// SIMATIC S7-200 project (STEP 7-Micro/WIN), CPU 226 CN REL 02.01

ORGANIZATION_BLOCK 主程序:OB1
TITLE=程序注释
BEGIN
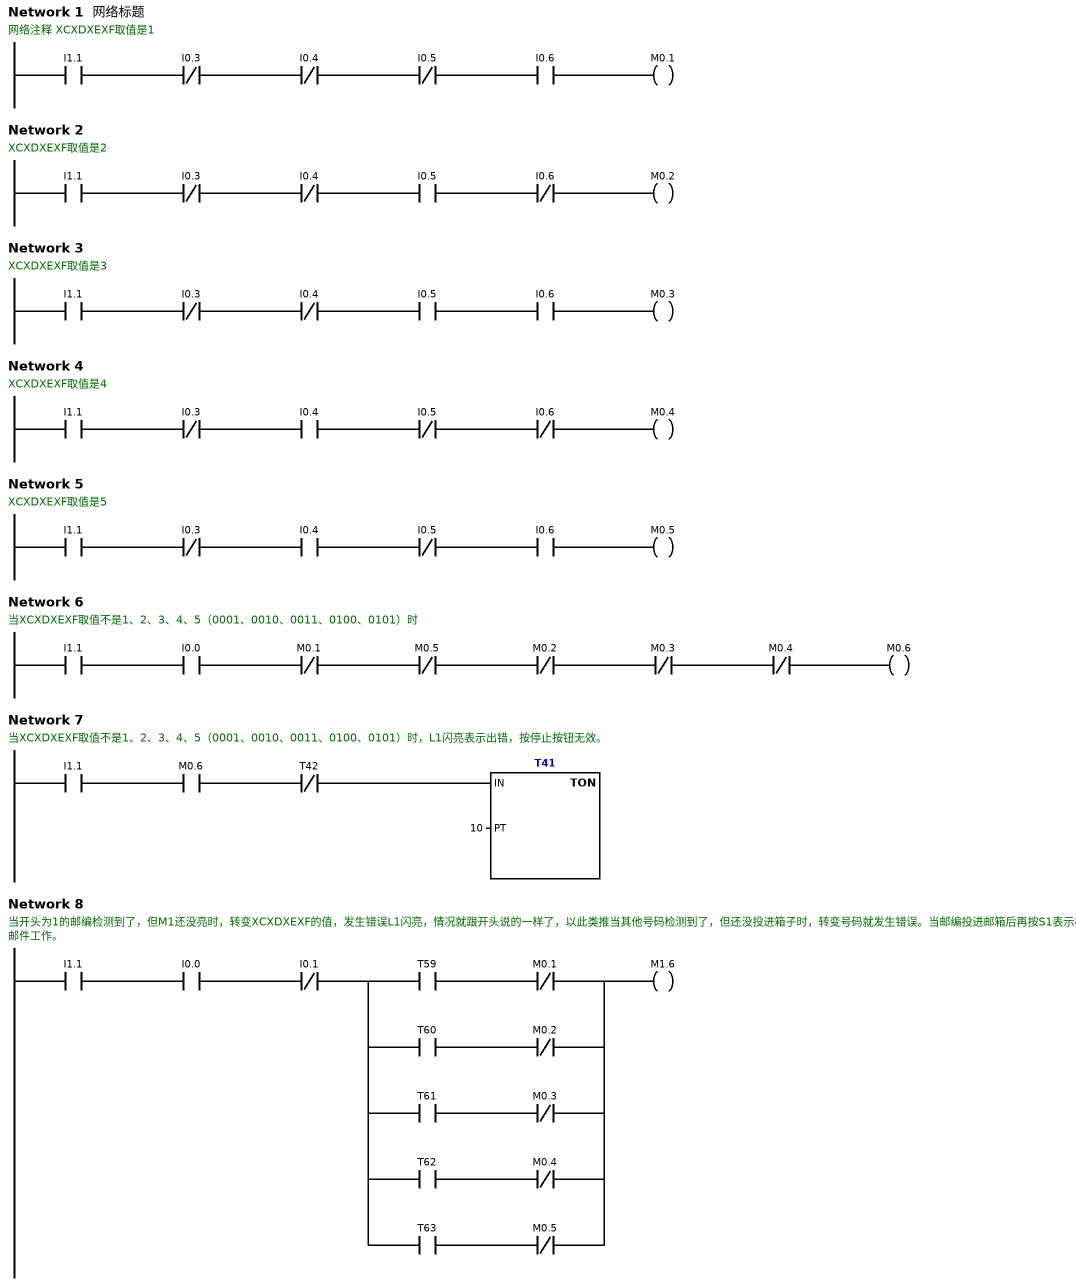
Network 1 // 网络标题
// 网络注释 XCXDXEXF取值是1
LD     I1.1
AN     I0.3
AN     I0.4
AN     I0.5
A      I0.6
=      M0.1
Network 2
// XCXDXEXF取值是2
LD     I1.1
AN     I0.3
AN     I0.4
A      I0.5
AN     I0.6
=      M0.2
Network 3
// XCXDXEXF取值是3
LD     I1.1
AN     I0.3
AN     I0.4
A      I0.5
A      I0.6
=      M0.3
Network 4
// XCXDXEXF取值是4
LD     I1.1
AN     I0.3
A      I0.4
AN     I0.5
AN     I0.6
=      M0.4
Network 5
// XCXDXEXF取值是5
LD     I1.1
AN     I0.3
A      I0.4
AN     I0.5
A      I0.6
=      M0.5
Network 6
// 当XCXDXEXF取值不是1、2、3、4、5（0001、0010、0011、0100、0101）时
LD     I1.1
A      I0.0
AN     M0.1
AN     M0.5
AN     M0.2
AN     M0.3
AN     M0.4
=      M0.6
Network 7
// 当XCXDXEXF取值不是1、2、3、4、5（0001、0010、0011、0100、0101）时，L1闪亮表示出错，按停止按钮无效。
LD     I1.1
A      M0.6
AN     T42
TON    T41, 10
Network 8
// 当开头为1的邮编检测到了，但M1还没亮时，转变XCXDXEXF的值，发生错误L1闪亮，情况就跟开头说的一样了，以此类推当其他号码检测到了，但还没投进箱子时，转变号码就发生错误。当邮编投进邮箱后再按S1表示检测到邮件工作。
// (network saved uncompiled; LAD cells follow)
// row 0: c0 -| |- I1.1  c1 -| |- I0.0  c2 -|/|- I0.1 v  c3 -| |- T59  c4 -|/|- M0.1 v  c5 -( ) M1.6
// row 1: c2 ^v  c3 -| |- T60  c4 -|/|- M0.2 ^v
// row 2: c2 ^v  c3 -| |- T61  c4 -|/|- M0.3 ^v
// row 3: c2 ^v  c3 -| |- T62  c4 -|/|- M0.4 ^v
// row 4: c2 ^  c3 -| |- T63  c4 -|/|- M0.5 ^
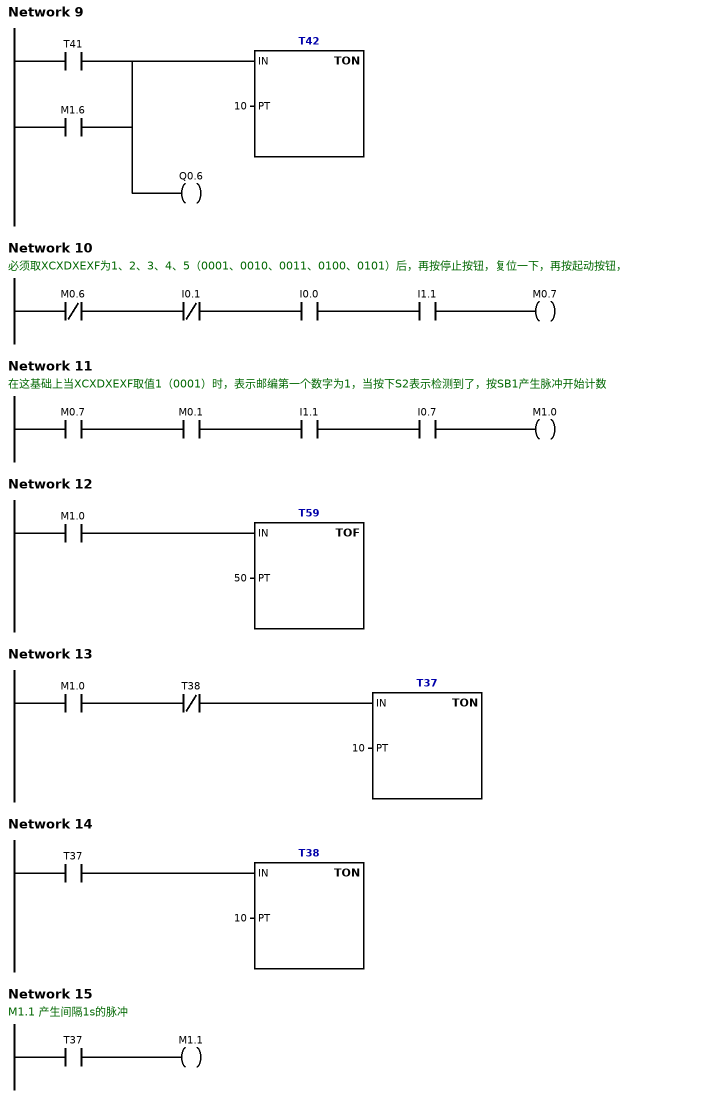
Network 9
LD     T41
O      M1.6
TON    T42, 10
=      Q0.6
Network 10
// 必须取XCXDXEXF为1、2、3、4、5（0001、0010、0011、0100、0101）后，再按停止按钮，复位一下，再按起动按钮，
LDN    M0.6
AN     I0.1
A      I0.0
A      I1.1
=      M0.7
Network 11
// 在这基础上当XCXDXEXF取值1（0001）时，表示邮编第一个数字为1，当按下S2表示检测到了，按SB1产生脉冲开始计数
LD     M0.7
A      M0.1
A      I1.1
A      I0.7
=      M1.0
Network 12
// (network saved uncompiled; LAD cells follow)
// row 0: c0 -| |- M1.0  c1 --  c2 [TOF T59 IN:=power@row0, PT:=50]
// row 1: c2 [box]
Network 13
LD     M1.0
AN     T38
TON    T37, 10
Network 14
LD     T37
TON    T38, 10
Network 15
// M1.1 产生间隔1s的脉冲
LD     T37
=      M1.1
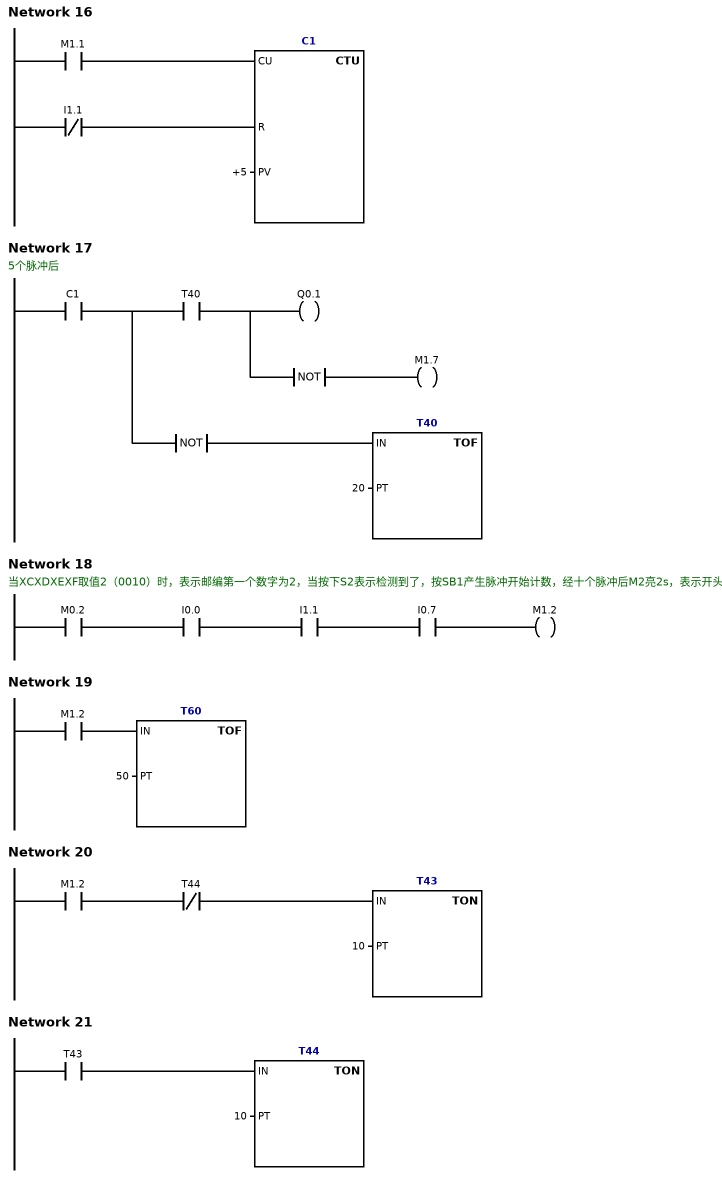
Network 16
LD     M1.1
LDN    I1.1
CTU    C1, +5
Network 17
// 5个脉冲后
LD     C1
LPS
A      T40
=      Q0.1
NOT
=      M1.7
LPP
NOT
TOF    T40, 20
Network 18
// 当XCXDXEXF取值2（0010）时，表示邮编第一个数字为2，当按下S2表示检测到了，按SB1产生脉冲开始计数，经十个脉冲后M2亮2s，表示开头为2的邮编进上海的邮箱，同时M5、L2、S1灭2s。
LD     M0.2
A      I0.0
A      I1.1
A      I0.7
=      M1.2
Network 19
// (network saved uncompiled; LAD cells follow)
// row 0: c0 -| |- M1.2  c1 [TOF T60 IN:=power@row0, PT:=50]
// row 1: c1 [box]
Network 20
LD     M1.2
AN     T44
TON    T43, 10
Network 21
LD     T43
TON    T44, 10
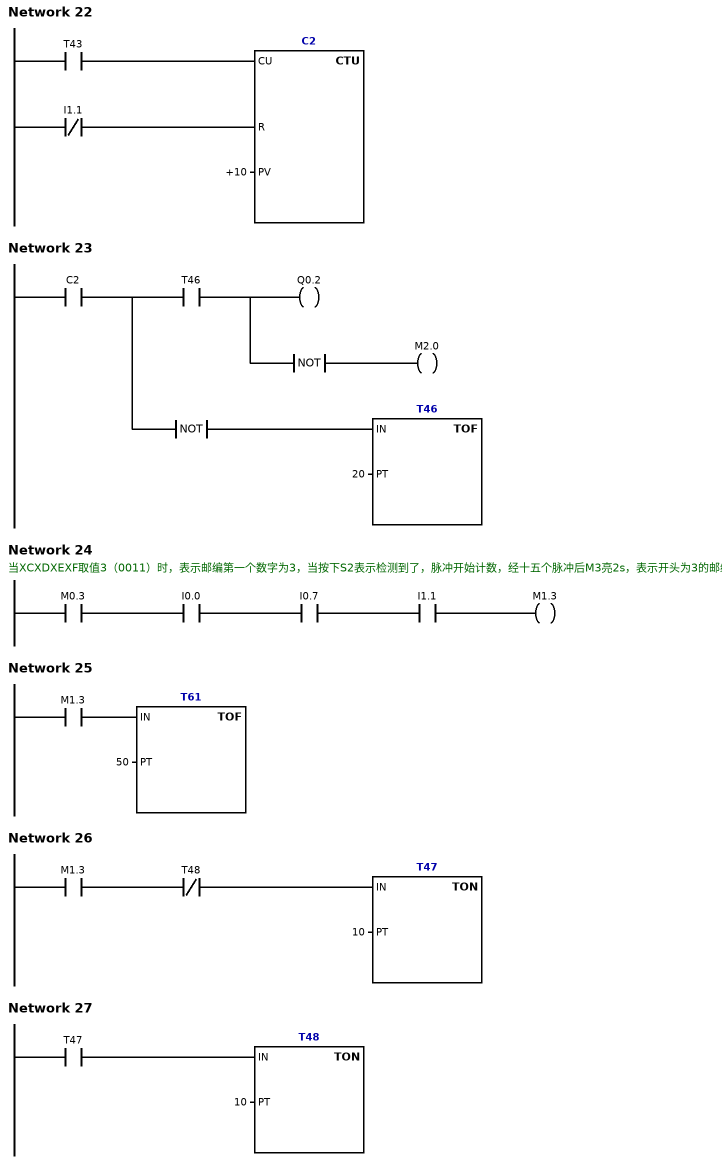
Network 22
LD     T43
LDN    I1.1
CTU    C2, +10
Network 23
LD     C2
LPS
A      T46
=      Q0.2
NOT
=      M2.0
LPP
NOT
TOF    T46, 20
Network 24
// 当XCXDXEXF取值3（0011）时，表示邮编第一个数字为3，当按下S2表示检测到了，脉冲开始计数，经十五个脉冲后M3亮2s，表示开头为3的邮编进天津的邮箱，同时M5、L2灭2s。
LD     M0.3
A      I0.0
A      I0.7
A      I1.1
=      M1.3
Network 25
// (network saved uncompiled; LAD cells follow)
// row 0: c0 -| |- M1.3  c1 [TOF T61 IN:=power@row0, PT:=50]
// row 1: c1 [box]
Network 26
LD     M1.3
AN     T48
TON    T47, 10
Network 27
LD     T47
TON    T48, 10
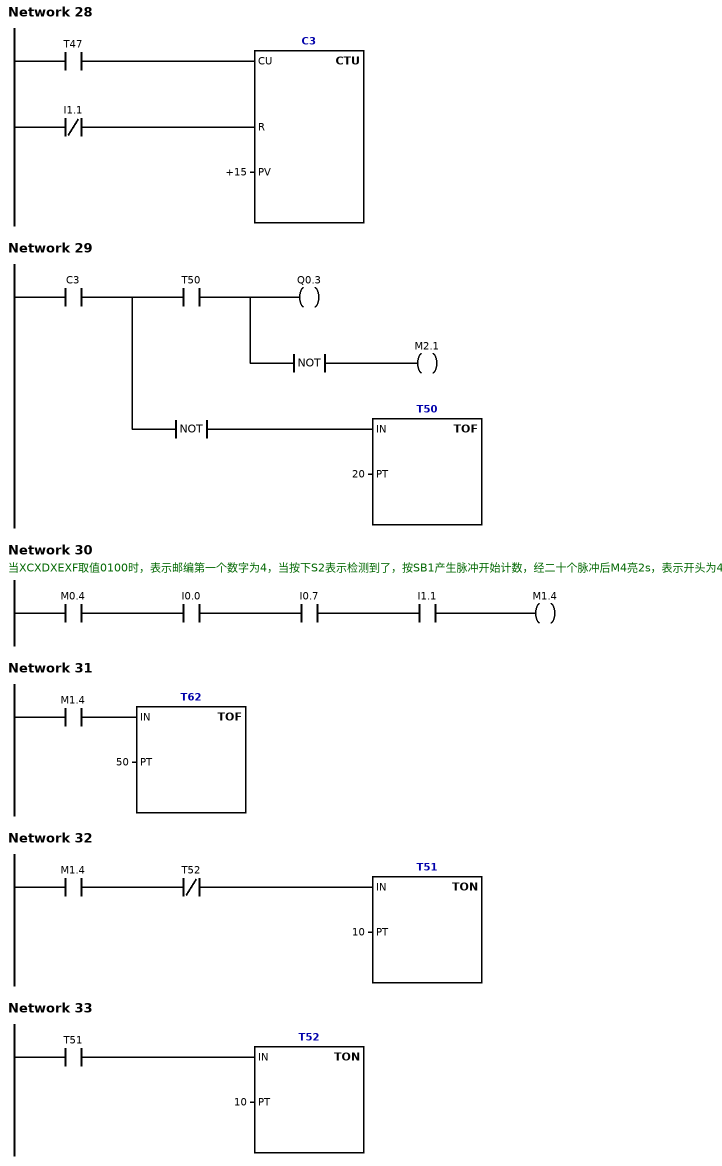
Network 28
LD     T47
LDN    I1.1
CTU    C3, +15
Network 29
LD     C3
LPS
A      T50
=      Q0.3
NOT
=      M2.1
LPP
NOT
TOF    T50, 20
Network 30
// 当XCXDXEXF取值0100时，表示邮编第一个数字为4，当按下S2表示检测到了，按SB1产生脉冲开始计数，经二十个脉冲后M4亮2s，表示开头为4的邮编进武汉的邮箱，同时M5、L2灭2s。
LD     M0.4
A      I0.0
A      I0.7
A      I1.1
=      M1.4
Network 31
// (network saved uncompiled; LAD cells follow)
// row 0: c0 -| |- M1.4  c1 [TOF T62 IN:=power@row0, PT:=50]
// row 1: c1 [box]
Network 32
LD     M1.4
AN     T52
TON    T51, 10
Network 33
LD     T51
TON    T52, 10
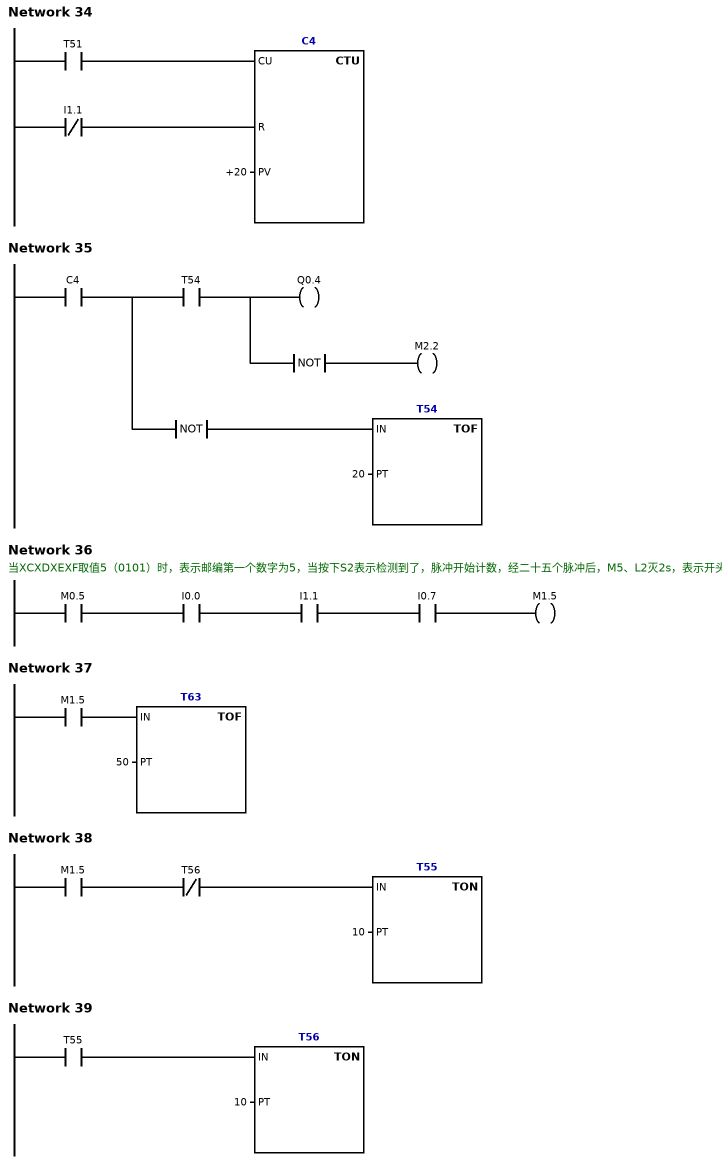
Network 34
LD     T51
LDN    I1.1
CTU    C4, +20
Network 35
LD     C4
LPS
A      T54
=      Q0.4
NOT
=      M2.2
LPP
NOT
TOF    T54, 20
Network 36
// 当XCXDXEXF取值5（0101）时，表示邮编第一个数字为5，当按下S2表示检测到了，脉冲开始计数，经二十五个脉冲后，M5、L2灭2s，表示开头为5的邮编进广州的邮箱。
LD     M0.5
A      I0.0
A      I1.1
A      I0.7
=      M1.5
Network 37
// (network saved uncompiled; LAD cells follow)
// row 0: c0 -| |- M1.5  c1 [TOF T63 IN:=power@row0, PT:=50]
// row 1: c1 [box]
Network 38
LD     M1.5
AN     T56
TON    T55, 10
Network 39
LD     T55
TON    T56, 10
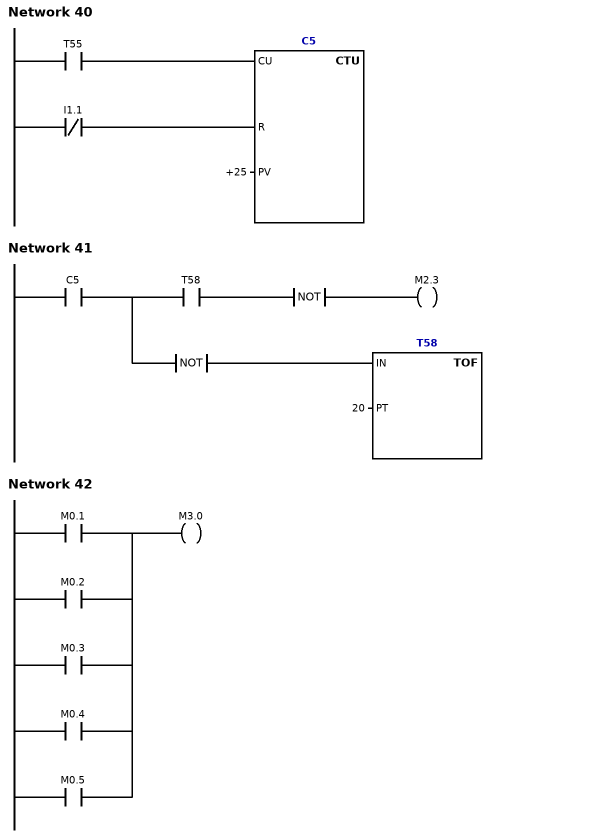
Network 40
LD     T55
LDN    I1.1
CTU    C5, +25
Network 41
LD     C5
LPS
A      T58
NOT
=      M2.3
LPP
NOT
TOF    T58, 20
Network 42
LD     M0.1
O      M0.2
O      M0.3
O      M0.4
O      M0.5
=      M3.0
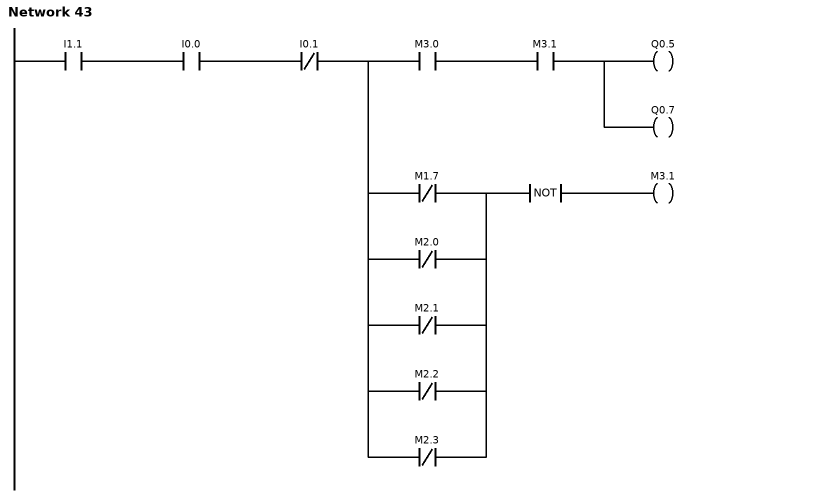
Network 43
LD     I1.1
A      I0.0
AN     I0.1
LPS
A      M3.0
A      M3.1
=      Q0.5
=      Q0.7
LPP
LDN    M1.7
ON     M2.0
ON     M2.1
ON     M2.2
ON     M2.3
ALD
NOT
=      M3.1
END_ORGANIZATION_BLOCK
